TYPE ST_ConveyorErrors :
STRUCT
	NCAxisError					: ST_NcAxis_Errors;
	
END_STRUCT
END_TYPE

(* stored: Version 1.1.0.1, ProductVersion 3.1.4020.12
   DUT ST_ConveyorErrors: Id {32c2723b-777b-4a73-bdcc-341715c91bd4} *)
